FUNCTION_BLOCK FB_CylinderSpringReturn IMPLEMENTS ICylinder
VAR
	Solenoid AT %Q* : BOOL;
END_VAR

METHOD Extend : BOOL
Solenoid := TRUE;
Extend	 := TRUE;
END_METHOD

METHOD Retract : BOOL
Solenoid := FALSE;
Retract	 := TRUE;
END_METHOD

END_FUNCTION_BLOCK

(* stored: Version 1.1.0.1, ProductVersion 3.1.4024.12
   POU FB_CylinderSpringReturn: Id {2e62cab7-a5c3-4da6-9737-990bfeb97ff9}, SpecialFunc None
   Method Extend: Id {42462696-ae31-4f4d-81a4-65ef9e89facd}
   Method Retract: Id {e92501ac-b2b9-4242-be88-4077c9a9f02f} *)
